PROGRAM PMPS
VAR
	
END_VAR

(*FastFaultOuput*)
g_FastFaultOutput1.Execute(bAutoReset:= TRUE);
g_FastFaultOutput2.Execute(i_xVeto:=PMPS_GVL.stCurrentBeamParameters.aStoppers[K_Stopper.ST1], bAutoReset:= TRUE);

END_PROGRAM

(* stored: Version 1.1.0.1, ProductVersion 3.1.4022.18
   POU PMPS: Id {354279ff-d518-454c-b9bb-5f6640e67b86}, SpecialFunc None *)
